screen "Screen_2" 800x480, template "KTP700 logo & menu"
   on GenerateScreen: SetTag("Screen_number", 2)
   Button "Button_1" at 14,122 size 55x55; TextOff '1'
      on Press: function_b14e0dd5("main_DB_Button_Screen_1_Z.P 1", 0)
      Appearance <- "Z.P 1"
   TextField "Text field_2" at 9,83 size 220x27; Text 'Zawory pnaumatyczne'
   TextField "Text field_3" at 350,84 size 266x34; Text 'Zawory hydrauliczne'
   Button "Button_2" at 14,179 size 55x55; TextOff '2'
      on Press: function_b14e0dd5("main_DB_Button_Screen_1_Z.P 2", 0)
      Appearance <- "Z.P 2"
   Button "Button_3" at 14,237 size 55x55; TextOff '3'
      on Press: function_b14e0dd5("main_DB_Button_Screen_1_Z.P 3", 0)
      Appearance <- "Z.P 3"
   Button "Button_4" at 14,295 size 55x55; TextOff '4'
      on Press: function_b14e0dd5("main_DB_Button_Screen_1_Z.P 4", 0)
      Appearance <- "Z.P 4"
   Button "Button_5" at 14,362 size 55x55; TextOff '0'
      on Press: function_b14e0dd5("main_DB_Button_Screen_1_Z.P 0", 0)
      Appearance <- "Z.P 0"
   Button "Button_10" at 254,122 size 55x55; TextOff '1'
      on Press: function_b14e0dd5("main_DB_Button_Screen_1_Z.H 1", 0)
      Appearance <- "Z.H 1"
   Button "Button_11" at 254,179 size 55x55; TextOff '3'
      on Press: function_b14e0dd5("main_DB_Button_Screen_1_Z.H 3", 0)
      Appearance <- "Z.H 3"
   Button "Button_12" at 254,237 size 55x55; TextOff '5'
      on Press: function_b14e0dd5("main_DB_Button_Screen_1_Z.H 5", 0)
      Appearance <- "Z.H 5"
   Button "Button_13" at 254,295 size 55x55; TextOff '7'
      on Press: function_b14e0dd5("main_DB_Button_Screen_1_Z.H 7", 0)
      Appearance <- "Z.H 7"
   Button "Button_14" at 254,362 size 55x55; TextOff '0'
      on Press: function_b14e0dd5("main_DB_Button_Screen_1_Z.H 0", 0)
      Appearance <- "Z.H 0"
   Button "Button_15" at 495,122 size 55x55; TextOff '2'
      on Press: function_b14e0dd5("main_DB_Button_Screen_1_Z.H 2", 0)
      Appearance <- "Z.H 2"
   Button "Button_16" at 495,179 size 55x55; TextOff '4'
      on Press: function_b14e0dd5("main_DB_Button_Screen_1_Z.H 4", 0)
      Appearance <- "Z.H 4"
   Button "Button_17" at 495,237 size 55x55; TextOff '6'
      on Press: function_b14e0dd5("main_DB_Button_Screen_1_Z.H 6", 0)
      Appearance <- "Z.H 6"
   Button "Button_18" at 495,295 size 55x55; TextOff '8'
      on Press: function_b14e0dd5("main_DB_Button_Screen_1_Z.H 8", 0)
      Appearance <- "Z.H 8"
   TextField "Text field_16" at 73,376 size 141x27; Text 'Zawór główny'
   TextField "Text field_17" at 313,376 size 141x27; Text 'Zawór główny'
   Button "Button_6" at 14,428 size 160x45; TextOff 'Sterowanie ręczne'
      on Press: function_b14e0dd5("main_DB_Button_Screen_1_Manual_control", 0)
      Appearance <- "main_DB_Status_Manual_control"
   Button "Button_7" at 292,428 size 160x45; TextOff 'Załączenie pompy hydraulicznej'
      on Press: function_b14e0dd5("main_DB_Button_Screen_1_Hydraulic_Pump", 0)
      Appearance <- "Pompa hydrauliczna"
   IOField "I/O field_1" at 72,134 size 156x32; FormatPattern ????????????????????????????????????????????????????????????????????????????????
      ProcessValue <- "main_DB_var_Descryption Z.P 1"
   IOField "I/O field_2" at 72,191 size 156x32; FormatPattern ????????????????????????????????????????????????????????????????????????????????
      ProcessValue <- "main_DB_var_Descryption Z.P 2"
   IOField "I/O field_3" at 72,249 size 156x32; FormatPattern ????????????????????????????????????????????????????????????????????????????????
      ProcessValue <- "main_DB_var_Descryption Z.P 3"
   IOField "I/O field_4" at 72,307 size 156x32; FormatPattern ????????????????????????????????????????????????????????????????????????????????
      ProcessValue <- "main_DB_var_Descryption Z.P 4"
   IOField "I/O field_5" at 313,134 size 156x32; FormatPattern ????????????????????????????????????????????????????????????????????????????????
      ProcessValue <- "main_DB_var_Descryption Z.H 1"
   IOField "I/O field_6" at 313,191 size 156x32; FormatPattern ????????????????????????????????????????????????????????????????????????????????
      ProcessValue <- "main_DB_var_Descryption Z.H 3"
   IOField "I/O field_7" at 313,249 size 156x32; FormatPattern ????????????????????????????????????????????????????????????????????????????????
      ProcessValue <- "main_DB_var_Descryption Z.H 5"
   IOField "I/O field_8" at 313,307 size 156x32; FormatPattern ????????????????????????????????????????????????????????????????????????????????
      ProcessValue <- "main_DB_var_Descryption Z.H 7"
   IOField "I/O field_9" at 554,134 size 156x32; FormatPattern ????????????????????????????????????????????????????????????????????????????????
      ProcessValue <- "main_DB_var_Descryption Z.H 2"
   IOField "I/O field_10" at 554,191 size 156x32; FormatPattern ????????????????????????????????????????????????????????????????????????????????
      ProcessValue <- "main_DB_var_Descryption Z.H 4"
   IOField "I/O field_11" at 554,249 size 156x32; FormatPattern ????????????????????????????????????????????????????????????????????????????????
      ProcessValue <- "main_DB_var_Descryption Z.H 6"
   IOField "I/O field_12" at 554,307 size 156x32; FormatPattern ????????????????????????????????????????????????????????????????????????????????
      ProcessValue <- "main_DB_var_Descryption Z.H 8"
   Button "Button_8" at 550,428 size 160x45; TextOff 'Odprężenie'
      on Press: function_b14e0dd5("main_DB_Button_Screen_2_Relaxation", 0)
      Appearance <- "main_DB_Status_relaxation"

screen "Screen_3" 800x480, template "KTP700 logo & menu"
   on GenerateScreen: SetTag("Screen_number", 3)
   Button "Button_1" at 14,122 size 55x55; TextOff '1'
      Appearance <- "SQ1"
   Button "Button_2" at 14,179 size 55x55; TextOff '2'
      Appearance <- "SQ2"
   Button "Button_3" at 14,237 size 55x55; TextOff '3'
      Appearance <- "SQ3"
   Button "Button_4" at 14,295 size 55x55; TextOff '4'
      Appearance <- "SQ4"
   Button "Button_5" at 14,353 size 55x55; TextOff '5'
      Appearance <- "SQ5"
   Button "Button_6" at 14,411 size 55x55; TextOff '6'
      Appearance <- "SQ6"
   Button "Button_7" at 382,122 size 55x55; TextOff '1'
      Appearance <- "zwierny_1"
   Button "Button_8" at 382,179 size 55x55; TextOff '2'
      Appearance <- "zwierny_2"
   Button "Button_9" at 382,237 size 55x55; TextOff '3'
      Appearance <- "zwierny_3"
   Button "Button_10" at 382,295 size 55x55; TextOff '4'
      Appearance <- "zwierny_4"
   Button "Button_11" at 382,353 size 55x55; TextOff '5'
      Appearance <- "zwierny_5"
   Button "Button_12" at 382,411 size 55x55; TextOff '6'
      Appearance <- "zwierny_6"
   IOField "I/O field_1" at 72,134 size 275x32; FormatPattern ????????????????????????????????????????????????????????????????????????????????
      ProcessValue <- "main_DB_var_Descryption SQ 1"
   IOField "I/O field_2" at 72,191 size 275x32; FormatPattern ????????????????????????????????????????????????????????????????????????????????
      ProcessValue <- "main_DB_var_Descryption SQ 2"
   IOField "I/O field_3" at 72,249 size 275x32; FormatPattern ????????????????????????????????????????????????????????????????????????????????
      ProcessValue <- "main_DB_var_Descryption SQ 3"
   IOField "I/O field_4" at 72,307 size 275x32; FormatPattern ????????????????????????????????????????????????????????????????????????????????
      ProcessValue <- "main_DB_var_Descryption SQ 4"
   IOField "I/O field_5" at 72,365 size 275x32; FormatPattern ????????????????????????????????????????????????????????????????????????????????
      ProcessValue <- "main_DB_var_Descryption SQ 5"
   IOField "I/O field_6" at 72,423 size 275x32; FormatPattern ????????????????????????????????????????????????????????????????????????????????
      ProcessValue <- "main_DB_var_Descryption SQ 6"
   IOField "I/O field_7" at 441,134 size 275x32; FormatPattern ????????????????????????????????????????????????????????????????????????????????
      ProcessValue <- "main_DB_var_Descryption contact_sensor 1"
   IOField "I/O field_8" at 441,191 size 275x32; FormatPattern ????????????????????????????????????????????????????????????????????????????????
      ProcessValue <- "main_DB_var_Descryption contact_sensor 2"
   IOField "I/O field_9" at 441,249 size 275x32; FormatPattern ????????????????????????????????????????????????????????????????????????????????
      ProcessValue <- "main_DB_var_Descryption contact_sensor 3"
   IOField "I/O field_10" at 441,307 size 275x32; FormatPattern ????????????????????????????????????????????????????????????????????????????????
      ProcessValue <- "main_DB_var_Descryption contact_sensor 4"
   IOField "I/O field_11" at 441,365 size 275x32; FormatPattern ????????????????????????????????????????????????????????????????????????????????
      ProcessValue <- "main_DB_var_Descryption contact_sensor 5"
   IOField "I/O field_12" at 441,423 size 275x32; FormatPattern ????????????????????????????????????????????????????????????????????????????????
      ProcessValue <- "main_DB_var_Descryption contact_sensor 6"
   TextField "Text field_3" at 0,85 size 364x34; Text 'Czujniki indukcyjne'
   TextField "Text field_1" at 358,85 size 367x34; Text 'Kołki stykowe'
*)